(* IEC 61131-3 sources: Industry-PLC-LLM/data/PLCBEAD_repo/PLCBEAD_PLCEmbed-main/PLC-BEAD/Source/GEB/TREND, 1 file *)

(* ---- TREND.ST ---- *)
FUNCTION_BLOCK TREND

	VAR_INPUT
		X :	REAL;
	END_VAR

	VAR_OUTPUT
		Q :	BOOL;
		TU :	BOOL;
		TD :	BOOL;
		D :	REAL;
	END_VAR

	VAR
		last_x :	REAL;
	END_VAR

	TU := X > last_X;
	TD := X < last_X;
	Q := TU OR TD;
	D := X - LAST_X;

	last_X := X;

END_FUNCTION_BLOCK

PROGRAM program0
  VAR
	X :	REAL;
	Q :	BOOL;
	TU :	BOOL;
	TD :	BOOL;
	D :	REAL;
	func_block : TREND;
  END_VAR
	func_block.X  :=X ;
	func_block();
	Q := func_block.Q;
	TU := func_block.TU;
	TD := func_block.TD;
	D := func_block.D;
END_PROGRAM
